Staubli VAL3: WriteSingIOMsg.pjx

--- WriteSingIOMsg.pjx ---
Parameters version=s7.9.1 stackSize=5000 millimeterUnit=true
Program file=start.pgx
Program file=stop.pgx
Data file=WriteSingIOMsg.dtx
Type name=Body path=Disk://ros_libs/Body/Body.pjx
Type name=Header path=Disk://ros_libs/Header/Header.pjx
Type name=Prefix path=Disk://ros_libs/Prefix/Prefix.pjx
Type name=WriteSingleIO path=../WriteSingleIO/WriteSingleIO.pjx

--- WriteSingIOMsg.dtx ---
public Body body
  [0]
    num nData[9]
public Header header
  [0]
    num nCommType
    num nData[12]
    num nMsgType
    num nReplyCode
public Prefix prefix
  [0]
    num nData[4]
    num nLength
public WriteSingleIO writeSingleIO
  [0]
    bool bState
    num nModuleId
    num nPin
